FUNCTION ISBOOLEAN : BOOL
VAR_INPUT
	In:		POINTER TO STRING(5);
END_VAR
VAR
	TempVar:	STRING(5);
END_VAR

(*=======================================================================================================
ISBOOLEAN()
Author: Tim Van Meppelen, Pro Electric Inc.
timv@proelectric.com
Date: Oct 2, 2018
check if a string would convert to a valid boolean variable
========================================================================================================*)
TempVar:= In^;
StrToUpperA(pString:= ADR(TempVar));

ISBOOLEAN:= (TempVar = 'TRUE') OR (TempVar = 'FALSE');

END_FUNCTION

(* stored: Version 1.1.0.1
   POU ISBOOLEAN: Id {90377328-7a8b-4e27-a839-20f33a43f549}, SpecialFunc None *)
